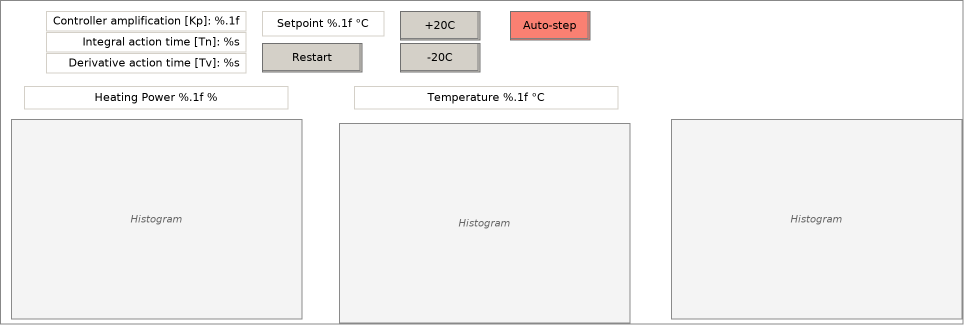
VISUALIZATION VIS_HEATER_CONTROL  // 964x325
    Histogram (11,119 291x200), scale format: %.1f, scale 0..100
        p1518820177: gstHistory.arPower
        p102497268: gstHistory.arPower
        p788070771: ARRAY [1..NUM_HISTORY_POINTS] OF REAL
    Histogram (339,123 291x200), scale format: %.1f, scale 0..200
        p1518820177: gstHistory.arTemperature
        p102497268: gstHistory.arTemperature
        p788070771: ARRAY [1..NUM_HISTORY_POINTS] OF REAL
    Textfield (24,86 264x23), "Heating Power %.1f %", text variable: gPower
    Textfield (354,86 264x23), "Temperature %.1f °C", text variable: IO_Inputs.i_HtrTemp
    Textfield (262,11 122x25), "Setpoint %.1f °C", text variable: gSetpoint
        OnMouseClick: write the text variable via Default
    Textfield (46,53 200x20), "Derivative action time [Tv]: %s", text variable: MAIN.fbHeaterCtrl.stParams.tTv
        OnMouseClick: write the text variable via Default
    Button (262,43 100x29), "Restart"
        tap IO_Outputs.o_Restart
    Textfield (46,32 200x20), "Integral action time [Tn]: %s", text variable: MAIN.fbHeaterCtrl.stParams.tTn
        OnMouseClick: write the text variable via Default
    Textfield (46,11 200x20), "Controller amplification [Kp]: %.1f", text variable: MAIN.fbHeaterCtrl.stParams.fKp
        OnMouseClick: write the text variable via Default
    Button (400,11 80x29), "+20C"
        tap IO_Outputs.o_AddTemp20
    Button (400,43 80x29), "-20C"
        tap IO_Outputs.o_DropTemp20
    Histogram (671,119 291x200), scale format: %.1f, scale -5..5
        p1518820177: gstHistory.arTempDiff
        p102497268: gstHistory.arTempDiff
        p788070771: ARRAY [1..NUM_HISTORY_POINTS] OF REAL
    Button (510,11 80x29), "Auto-step", colour toggle: gBoolAutoStep
        tap IO_Outputs.o_AutoStep
END_VISUALIZATION

(* stored: Version 1.1.0.1, ProductVersion 3.1.4022.18
   Visu VIS_HEATER_CONTROL: Id {053f00c4-a77d-4e3f-8faf-59312a40128a} *)
